FUNCTION_BLOCK FB_ModBus_100Registers_FC3
VAR_INPUT PERSISTENT
	m_Enable					: BOOL;						//Enable the Fuctionblock and his logic
	str_IPAdress				: STRING(15);				//IP Adress of the meter
	w_Adress					: WORD;						//modbus adress
	usint_Quantity				: usINT;						//Number of Words to get polled, max 100
END_VAR
VAR_OUTPUT
	m_PollSuccessful			: BOOL;						//Poll succesfull		
	w_Array_Received			: ARRAY[1..100] OF WORD;	// received data
	udint_Error_ID				: UDINT;					// ERR ID FB_MBReadRegs
END_VAR
VAR
	
	timer_Delay					: TON;						//Timer for Delay between Requests
	
	timer_DelayStart			: TON;						//Timer to start the state machine with Delay after enabling or after the system ist restartet
	
	timer_TimeOut				: TON;						//Timer for Timeout MB Read
	
	iStateModbusRead			: INT;						//State machine for read out Data over Modbus RTU
	
	fbMBRead_FC3				: FB_MBReadRegs  ;		//Modbus Read Function (FC3)
	
	ftrig_PEnable				: f_trig;					//Internal positive Edge
	
	iStateModbusError			: INT;						//State machine for error out Data over Modbus TCP/IP	
	
	FPError_FC_3				: R_TRIG;					//Internal positive Edge
	
	arrBuffer_FC3				: ARRAY[1..100] OF WORD;		//Buffer with Data from FC3
	
	timer_Connection_ok			: TON;
	int_Data_Received			: INT;
	
	m_MBTCPError				: BOOL;
	
	int_Data_Received_old		: INT;
	
	timer_Connection_ok_TOF	: TOF;
	
	fbConvertWordToDword		: FB_CV_WORD_TO_DWORD;			//Convert Word to Dword
	
	m_Poll_ok: BOOL;
	
	timer_Wait: Ton;
	int_TimeoutError: INT;
	int_FC3Error: INT;

END_VAR

(*	{attribute 'hide'}--------------------------------------------------------------------------------------------Limits-------------------------------------------------------------------------------------*)

w_Adress := LIMIT(0,w_Adress,60000);
usint_Quantity := LIMIT(1,usint_Quantity,100);
	
(*--------------------------------------------------------------------------------------------State Machine Read--------------------------------------------------------------------------------------*)

//Timer for Delay
timer_Delay(IN:= , PT:= T#50MS, Q=> , ET=> );

//Timeout Timer is dissabled when the Init Step is aktiv or the function is not enabled
IF iStateModbusRead = 0 OR NOT m_Enable THEN 
	timer_Timeout.IN := FALSE; 
END_IF
timer_Timeout(IN:= , PT:= T#1S, Q=> , ET=> );

//Enable with Delay that not all sockets have to be created at the same time
timer_DelayStart(IN:= m_Enable, PT:= T#1S, Q=> , ET=> );
ftrig_PEnable(CLK:= timer_DelayStart.Q, Q=> );

IF ftrig_PEnable.Q AND iStateModbusRead = 0 THEN 
	iStateModbusRead := 1; 
END_IF		
		
//Not Enabled
IF NOT m_Enable THEN 
	iStateModbusRead := 0; 
	iStateModbusError := 0; 
END_IF		
		
CASE iStateModbusRead OF

	0://Init Step 
		timer_Delay.IN := FALSE;
		fbMBRead_FC3.bExecute := FALSE;
		m_Poll_ok:=FALSE;
		int_Data_Received:=0;
	
		iStateModbusRead := 1;
	
	1://read the required registers
		//Start Read
		fbMBRead_FC3.nQuantity := usint_Quantity;
		fbMBRead_FC3.nMBAddr := w_Adress;
		fbMBRead_FC3.bExecute := TRUE;
		fbMBRead_FC3.nUnitID := 1;
		timer_Timeout.IN := TRUE;
		IF fbMBRead_FC3.bBusy THEN 
			timer_Delay.IN := TRUE; 
		END_IF
		
		//Wait for Delay, copy Data and then next step
		IF NOT fbMBRead_FC3.bBusy AND NOT fbMBRead_FC3.bError AND timer_Delay.Q THEN
			m_Poll_ok:=TRUE;
			int_Data_Received:=int_Data_Received+1;
			m_MBTCPError := FALSE; 
			
			w_Array_Received := arrBuffer_FC3;
			
			
			//Go to Next Step
			timer_Timeout.IN := FALSE;
			fbMBRead_FC3.bExecute := FALSE;
			timer_Delay.IN := FALSE;		
			iStateModbusRead := 3;
		END_IF	

		//Error or Timeout
		IF FPError_FC_3.Q THEN 
			iStateModbusError := 300;
			int_FC3Error := int_FC3Error+1;
		ELSIF timer_Timeout.Q THEN  
			timer_Timeout.IN := FALSE; 	
			iStateModbusError := 300;
			int_TimeoutError := int_TimeoutError+1;
		END_IF
		
	
	3://Wait and go to step 1
		//1 because 0 is the Init Step for Read
		timer_Wait.IN := TRUE;
		
		IF timer_Wait.Q = TRUE THEN
			iStateModbusRead := 1;
			timer_Wait.IN :=FALSE;
		END_IF

			
		
		//Error on Master, changes on Inputs or Timeout
		IF timer_Timeout.Q THEN 
			iStateModbusError := 300; 
		END_IF
	
END_CASE

(* wait timer*)

timer_Wait(PT:=T#3S);


(*------------------------------------------------------------------Error and Warning----------------------------------------------------------------------------*)	
 
timer_Connection_ok			(In:=int_Data_Received<>int_Data_Received_old,PT:=T#10S);
timer_Connection_ok_TOF		(In:=NOT(int_Data_Received<>int_Data_Received_old) AND int_Data_Received>3 ,PT:=T#20S);
int_Data_Received_old:=int_Data_Received;
m_PollSuccessful:=NOT timer_Connection_ok.Q AND timer_Connection_ok_TOF.Q ;

(*------------------------------------------------------------------------------------------Modbus TCP Functions---------------------------------------------------------------------------------------------*)

fbMBRead_FC3(	sIPAddr:= str_IPAdress, 
				nTCPPort:= 502,
				cbLength:= SIZEOF(arrBuffer_FC3), 
				pDestAddr:= ADR(arrBuffer_FC3), 
				tTimeout:= T#10S,
				nErrId => udint_Error_ID);

FPError_FC_3(CLK:= fbMBRead_FC3.bError, Q=> );		

(*------------------------------------------------------------------------------------------State Machine Error---------------------------------------------------------------------------------------------*)	

CASE iStateModbusError OF
	
	300://Error
		timer_Wait.IN :=TRUE;
		timer_Delay.IN := FALSE;
		fbMBRead_FC3.bExecute := FALSE;
		m_MBTCPError := TRUE; 		
		m_Poll_ok:=FALSE;
		int_Data_Received:=0;
				//Restart from new with the Read out part after an Error
		IF timer_Wait.Q = TRUE THEN
			iStateModbusRead := 0;	
			iStateModbusError := 0;
			timer_Wait.IN :=FALSE;
			timer_Timeout.IN := FALSE;
		END_IF		
							
END_CASE

END_FUNCTION_BLOCK

(* stored: Version 1.1.0.1, ProductVersion 3.1.4024.11
   POU FB_ModBus_100Registers_FC3: Id {daf436b8-b751-4d6b-b234-9be79388468a}, SpecialFunc None *)
